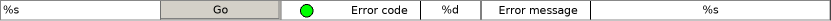
VISUALIZATION VISU_AlpacaPutRequest  // 831x21
VAR_IN_OUT
	stInstance : ST_AlpacaPutRequest;
END_VAR
    Rectangle (0,0 161x20), "%s", text variable: stInstance.sName
    Ellipse (300,4 13x13), colour toggle: stInstance.eStatusCode <> E_AlpacaStatusCode.OK
        p4168582468: stInstance.eStatusCode
    Button (160,0 121x20), "Go"
        OnMouseClick: execute { stInstance.bExecute := TRUE; }
    Label (350,0 61x21), "Error code"
    Rectangle (420,0 61x20), "%d", text variable: stInstance.nErrorCode
    Rectangle (590,0 241x20), "%s", text variable: stInstance.sErrorMessage
        p4168582468: stInstance.sErrorMessage
    Label (490,0 91x21), "Error message"
END_VISUALIZATION

(* stored: Version 1.1.0.1, ProductVersion 3.1.4024.12
   Visu VISU_AlpacaPutRequest: Id {159134cc-a4e7-4e95-9aa5-9821e61f19fa} *)
